# EPICS substitutions: iocbio4/iocBoot/UNUSED/canberra_3.substitutions
file "$(MCA)/mcaApp/Db/simple_mca.db"
{
pattern
{P           M       DTYP           INP              PREC  CHANS}
{18IDd:med:   mca1  "asynMCA"       "@asyn(AIM1/1 0)"  3     2048}
{18IDd:med:   mca2  "asynMCA"       "@asyn(AIM1/2 0)"  3     2048}
{18IDd:med:   mca3  "asynMCA"       "@asyn(AIM2/1 0)"  3     2048}
{18IDd:med:   mca0  "Soft Channel"  ""                 3     2048}
}

#file "$(MCA)/mcaApp/Db/icb_amp.db"
#{
#pattern
#{P			AMP		PORT}
#{18IDd:med:	amp1	icbAmp1}
#}

file "$(MCA)/mcaApp/Db/icb_adc.db"
{
pattern
{P			ADC		PORT}
{18IDd:med:	adc1	"icbAdc1"}
{18IDd:med:	adc2	"icbAdc2"}
{18IDd:med:	adc3	"icbAdc3"}
}

#file "$(MCA)/mcaApp/Db/icb_hvps.db"
#{
#pattern
#{P			HVPS	LIMIT	PORT}
#{18IDd:med:	hvps1	1000	"icbHvps1"}
#}

file "$(MCA)/mcaApp/Db/icb_tca.db"
{
pattern
{P,          TCA,	PORT,		MCA}
{18IDd:med:,  tca1,	"icbTca1",	mca1}
{18IDd:med:,  tca2,	"icbTca2",	mca2}
{18IDd:med:,  tca3,	"icbTca3",	mca3}
}
